{attribute 'linkalways'} 
{attribute 'no_explicit_call' := 'This FB is a CLASS and must be accessed using methods or properties'}
{attribute 'enable_dynamic_creation'}
FUNCTION_BLOCK INTERNAL MoveVelocityCommand EXTENDS MoveCommand
VAR
	_fb : MC_MoveVelocity;
END_VAR

METHOD FB_init : BOOL
VAR_INPUT
	bInitRetains : BOOL; // if TRUE, the retain variables are initialized (warm start / cold start)
	bInCopyCode : BOOL;  // if TRUE, the instance afterwards gets moved into the copy code (online change)
	axis : I_Axis;
	velocity : LREAL;
	acceleration : LREAL;
	deceleration : LREAL;
	jerk : LREAL;
	bufferMode : AxisBufferMode;
END_VAR
_axis := axis;
_velocity := velocity;
_acceleration := acceleration;
_deceleration := deceleration;
_jerk := jerk;
_bufferMode := bufferMode;
END_METHOD

METHOD PROTECTED WhileBusy
VAR_INPUT
	CommandState : I_CommandBusyState;
END_VAR
_fb(
	Axis := _axis._InternalAxisRef,
	Execute := TRUE,
	Velocity := _velocity,
	Acceleration := _acceleration,
	Deceleration := _deceleration,
	Jerk := _jerk,
	BufferMode := _bufferMode
);

IF _fb.Busy THEN
	RETURN;
END_IF

IF _fb.CommandAborted THEN
	_fb(Axis := _axis._InternalAxisRef, Execute := FALSE);
	CommandState.SetAborting();
	RETURN;
END_IF

IF _fb.Error THEN
	_fb(Axis := _axis._InternalAxisRef, Execute := FALSE);
	CommandState.SetError(_fb.ErrorID);
	RETURN;
END_IF

_fb(Axis := _axis._InternalAxisRef, Execute := FALSE);
CommandState.SetDone();
END_METHOD

END_FUNCTION_BLOCK

(* stored: Version 1.1.0.1, ProductVersion 3.1.4024.12
   POU MoveVelocityCommand: Id {b7ef6bbd-677a-4a49-9732-7d6bdc2cffe8}, SpecialFunc None
   Folder Constructor: Id {9f167e26-87ad-4e45-88bb-635a3e14b8fd}
   Method FB_init: Id {05ce250b-772e-48da-93e3-13b833c254d3}
   Method WhileBusy: Id {9339af6b-18d8-4c9e-a691-9cd16e0e009b} *)
